PROGRAM UnitTest
VAR
	fbTaskRunner_Test : FB_TaskRunner_Test;
	fbConveyorControl_Test : FB_ConveyorControl_Test;
	fbEventMessageQueue_Test : FB_EventMessageQueue_Test;
	fbFutureSleep_Test : FB_FutureSleep_Test;
	fbExecutor_Test : FB_Executor_Test;
END_VAR

// Production program — always runs regardless of variant
PRG_Conveyor();

{IF NOT defined (Release)}
fbTaskRunner_Test();
fbConveyorControl_Test();
fbEventMessageQueue_Test();
fbFutureSleep_Test();
fbExecutor_Test();
TcUnit.RUN();
{END_IF}

END_PROGRAM

(* stored: Version 1.1.0.1, ProductVersion 3.1.4024.15
   POU UnitTest: Id {3459d50f-46c2-4d8b-9955-5e66ae56a75a}, SpecialFunc None *)
